FUNCTION_BLOCK FB_StageRotate
VAR_INPUT
	bExecute		: BOOL;
END_VAR
VAR_OUTPUT
	bDone			: BOOL;
	bError			: BOOL;
	wErrorID		: BOOL;
END_VAR
VAR
	G1				: AXIS_REF;
	PowerOnG1		: MC_Power;
	PowerOnG1Out	: ST_McOutputs;
	ResetG1			: MC_Reset;
	ResetG1Out		: ST_McOutputs;
	HaltG1			: MC_Halt;
	HaltG1Out		: ST_McOutputs;
	HomeG1			: MC_Home;
	homeG1Out		: ST_McOutputs;
	JogG1			: MC_Jog;
	JogG1Out		: ST_McOutputs;
	MoveRelG1		: MC_MoveRelative;
	MoveRelG1Out		: ST_McOutputs;
END_VAR

G1();




actInit();
actMove();

ACTION actInit:
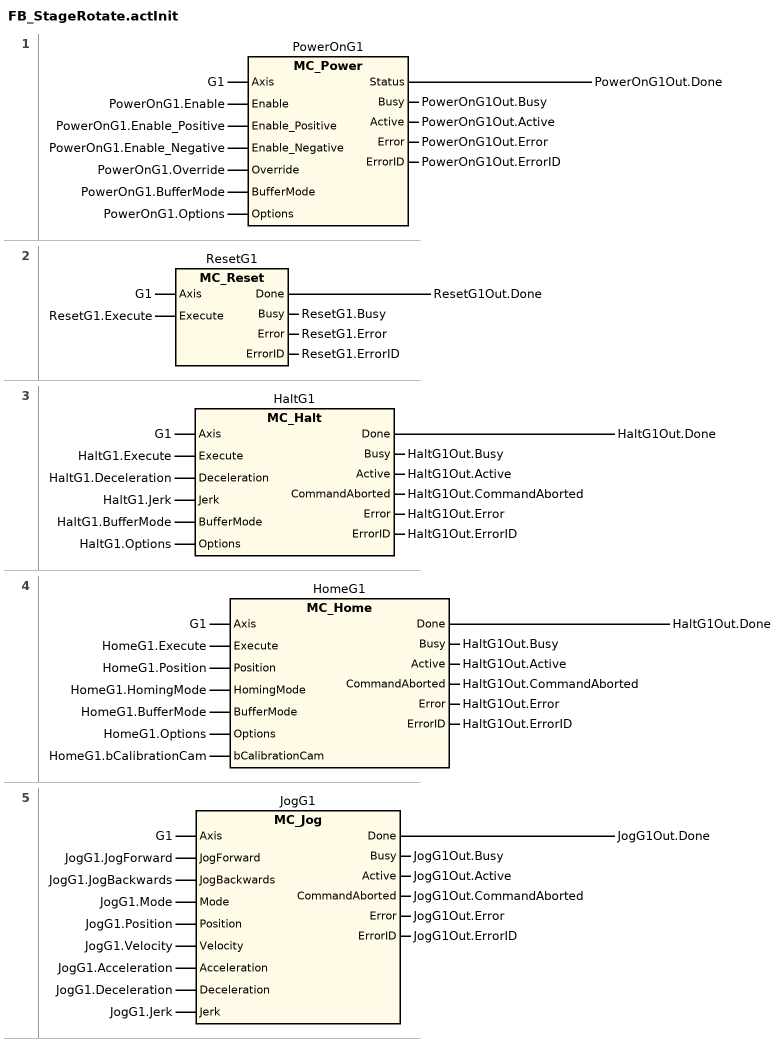
// NETWORK 1
PowerOnG1(
    Axis := G1,
    Enable := PowerOnG1.Enable,
    Enable_Positive := PowerOnG1.Enable_Positive,
    Enable_Negative := PowerOnG1.Enable_Negative,
    Override := PowerOnG1.Override,
    BufferMode := PowerOnG1.BufferMode,
    Options := PowerOnG1.Options,
    Busy => PowerOnG1Out.Busy,
    Active => PowerOnG1Out.Active,
    Error => PowerOnG1Out.Error,
    ErrorID => PowerOnG1Out.ErrorID); // MC_Power
PowerOnG1Out.Done := PowerOnG1.Status;

// NETWORK 2
ResetG1(
    Axis := G1,
    Execute := ResetG1.Execute,
    Busy => ResetG1.Busy,
    Error => ResetG1.Error,
    ErrorID => ResetG1.ErrorID); // MC_Reset
ResetG1Out.Done := ResetG1.Done;

// NETWORK 3
HaltG1(
    Axis := G1,
    Execute := HaltG1.Execute,
    Deceleration := HaltG1.Deceleration,
    Jerk := HaltG1.Jerk,
    BufferMode := HaltG1.BufferMode,
    Options := HaltG1.Options,
    Busy => HaltG1Out.Busy,
    Active => HaltG1Out.Active,
    CommandAborted => HaltG1Out.CommandAborted,
    Error => HaltG1Out.Error,
    ErrorID => HaltG1Out.ErrorID); // MC_Halt
HaltG1Out.Done := HaltG1.Done;

// NETWORK 4
HomeG1(
    Axis := G1,
    Execute := HomeG1.Execute,
    Position := HomeG1.Position,
    HomingMode := HomeG1.HomingMode,
    BufferMode := HomeG1.BufferMode,
    Options := HomeG1.Options,
    bCalibrationCam := HomeG1.bCalibrationCam,
    Busy => HaltG1Out.Busy,
    Active => HaltG1Out.Active,
    CommandAborted => HaltG1Out.CommandAborted,
    Error => HaltG1Out.Error,
    ErrorID => HaltG1Out.ErrorID); // MC_Home
HaltG1Out.Done := HomeG1.Done;

// NETWORK 5
JogG1(
    Axis := G1,
    JogForward := JogG1.JogForward,
    JogBackwards := JogG1.JogBackwards,
    Mode := JogG1.Mode,
    Position := JogG1.Position,
    Velocity := JogG1.Velocity,
    Acceleration := JogG1.Acceleration,
    Deceleration := JogG1.Deceleration,
    Jerk := JogG1.Jerk,
    Busy => JogG1Out.Busy,
    Active => JogG1Out.Active,
    CommandAborted => JogG1Out.CommandAborted,
    Error => JogG1Out.Error,
    ErrorID => JogG1Out.ErrorID); // MC_Jog
JogG1Out.Done := JogG1.Done;
END_ACTION

ACTION actMove:
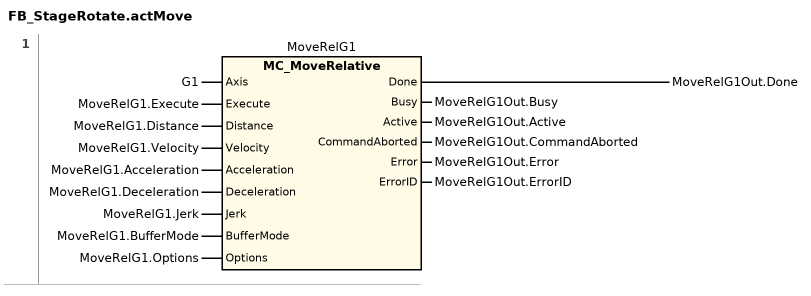
// NETWORK 1
MoveRelG1(
    Axis := G1,
    Execute := MoveRelG1.Execute,
    Distance := MoveRelG1.Distance,
    Velocity := MoveRelG1.Velocity,
    Acceleration := MoveRelG1.Acceleration,
    Deceleration := MoveRelG1.Deceleration,
    Jerk := MoveRelG1.Jerk,
    BufferMode := MoveRelG1.BufferMode,
    Options := MoveRelG1.Options,
    Busy => MoveRelG1Out.Busy,
    Active => MoveRelG1Out.Active,
    CommandAborted => MoveRelG1Out.CommandAborted,
    Error => MoveRelG1Out.Error,
    ErrorID => MoveRelG1Out.ErrorID); // MC_MoveRelative
MoveRelG1Out.Done := MoveRelG1.Done;
END_ACTION

END_FUNCTION_BLOCK

(* stored: Version 1.1.0.1, ProductVersion 3.1.4024.11
   POU FB_StageRotate: Id {97b2cf82-35e3-4a26-b77c-d043517303d6}, SpecialFunc None
   Action actInit: Id {f4bd0a5c-42a0-4a6e-ae3f-5b0f6ed6a683}
   Action actMove: Id {109d553b-ffa6-4d21-8812-231a0cde00c1} *)
